FUNCTION_BLOCK LoggerADS IMPLEMENTS I_Logger

METHOD trace
VAR_INPUT
	message	: T_MAXSTRING;
END_VAR
 ADSLOGSTR(msgCtrlMask := ADSLOG_MSGTYPE_HINT, msgFmtStr := message, strArg := '');
END_METHOD

END_FUNCTION_BLOCK

(* stored: Version 1.1.0.1, ProductVersion 3.1.4026.18
   POU LoggerADS: Id {7d8366ed-f454-4534-b8f1-0732cac7bf2c}, SpecialFunc None
   Method trace: Id {f7e97f75-c3ef-4d1b-96b4-9e73a98a8ea2} *)
